// TIA Portal V19 export
FUNCTION "Flowmeter Diag" : Void   // FC10, LAD
{ S7_Optimized_Access := 'TRUE' }
// stored: SetENOAutomatically false
BEGIN

REGION Network 1
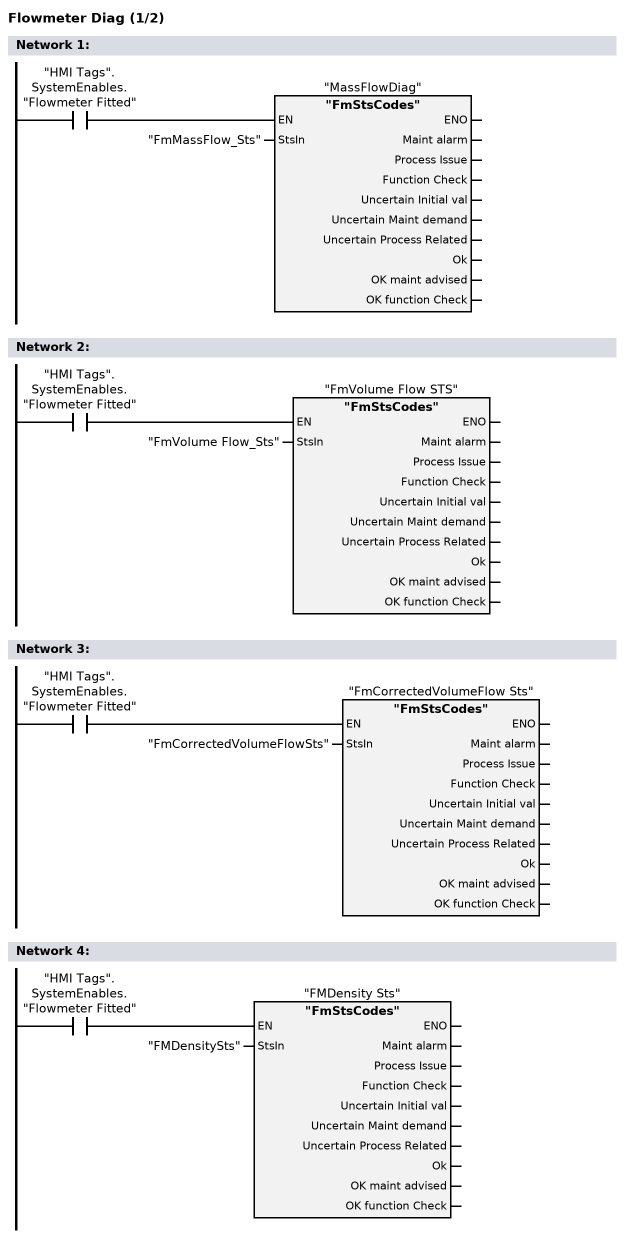
   RUNG wire#powerrail
      Contact( "HMI Tags".SystemEnables."Flowmeter Fitted" )
      "MassFlowDiag"(StsIn := "FmMassFlow_Sts", "Maint alarm" =>, "Process Issue" =>, "Function Check" =>, "Uncertain Initial val" =>, "Uncertain Maint demand" =>, "Uncertain Process Related" =>, Ok =>, "OK maint advised" =>, "OK function Check" =>)
   END_RUNG
   // the same network as SCL:
   IF "HMI Tags".SystemEnables."Flowmeter Fitted" THEN
       "MassFlowDiag"(StsIn := "FmMassFlow_Sts");   // "FmStsCodes"
   END_IF;
END_REGION

REGION Network 2
   RUNG wire#powerrail
      Contact( "HMI Tags".SystemEnables."Flowmeter Fitted" )
      "FmVolume Flow STS"(StsIn := "FmVolume Flow_Sts", "Maint alarm" =>, "Process Issue" =>, "Function Check" =>, "Uncertain Initial val" =>, "Uncertain Maint demand" =>, "Uncertain Process Related" =>, Ok =>, "OK maint advised" =>, "OK function Check" =>)
   END_RUNG
   // the same network as SCL:
   IF "HMI Tags".SystemEnables."Flowmeter Fitted" THEN
       "FmVolume Flow STS"(StsIn := "FmVolume Flow_Sts");   // "FmStsCodes"
   END_IF;
END_REGION

REGION Network 3
   RUNG wire#powerrail
      Contact( "HMI Tags".SystemEnables."Flowmeter Fitted" )
      "FmCorrectedVolumeFlow Sts"(StsIn := "FmCorrectedVolumeFlowSts", "Maint alarm" =>, "Process Issue" =>, "Function Check" =>, "Uncertain Initial val" =>, "Uncertain Maint demand" =>, "Uncertain Process Related" =>, Ok =>, "OK maint advised" =>, "OK function Check" =>)
   END_RUNG
   // the same network as SCL:
   IF "HMI Tags".SystemEnables."Flowmeter Fitted" THEN
       "FmCorrectedVolumeFlow Sts"(StsIn := "FmCorrectedVolumeFlowSts");   // "FmStsCodes"
   END_IF;
END_REGION

REGION Network 4
   RUNG wire#powerrail
      Contact( "HMI Tags".SystemEnables."Flowmeter Fitted" )
      "FMDensity Sts"(StsIn := "FMDensitySts", "Maint alarm" =>, "Process Issue" =>, "Function Check" =>, "Uncertain Initial val" =>, "Uncertain Maint demand" =>, "Uncertain Process Related" =>, Ok =>, "OK maint advised" =>, "OK function Check" =>)
   END_RUNG
   // the same network as SCL:
   IF "HMI Tags".SystemEnables."Flowmeter Fitted" THEN
       "FMDensity Sts"(StsIn := "FMDensitySts");   // "FmStsCodes"
   END_IF;
END_REGION

REGION Network 5
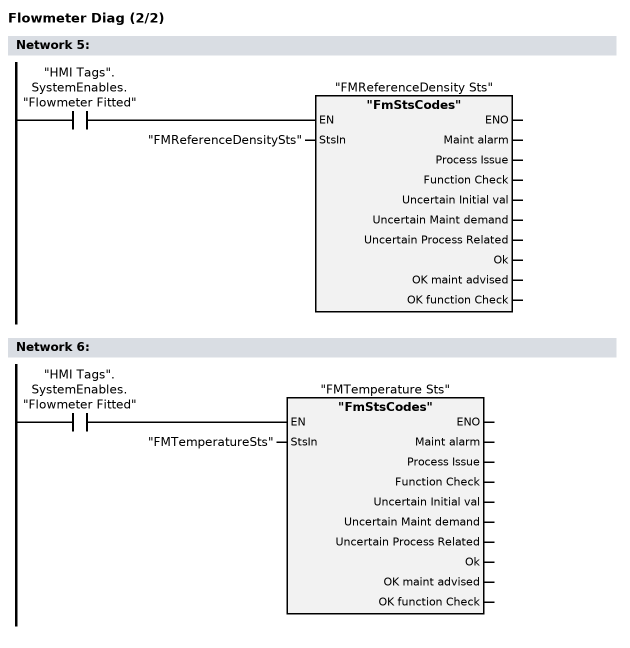
   RUNG wire#powerrail
      Contact( "HMI Tags".SystemEnables."Flowmeter Fitted" )
      "FMReferenceDensity Sts"(StsIn := "FMReferenceDensitySts", "Maint alarm" =>, "Process Issue" =>, "Function Check" =>, "Uncertain Initial val" =>, "Uncertain Maint demand" =>, "Uncertain Process Related" =>, Ok =>, "OK maint advised" =>, "OK function Check" =>)
   END_RUNG
   // the same network as SCL:
   IF "HMI Tags".SystemEnables."Flowmeter Fitted" THEN
       "FMReferenceDensity Sts"(StsIn := "FMReferenceDensitySts");   // "FmStsCodes"
   END_IF;
END_REGION

REGION Network 6
   RUNG wire#powerrail
      Contact( "HMI Tags".SystemEnables."Flowmeter Fitted" )
      "FMTemperature Sts"(StsIn := "FMTemperatureSts", "Maint alarm" =>, "Process Issue" =>, "Function Check" =>, "Uncertain Initial val" =>, "Uncertain Maint demand" =>, "Uncertain Process Related" =>, Ok =>, "OK maint advised" =>, "OK function Check" =>)
   END_RUNG
   // the same network as SCL:
   IF "HMI Tags".SystemEnables."Flowmeter Fitted" THEN
       "FMTemperature Sts"(StsIn := "FMTemperatureSts");   // "FmStsCodes"
   END_IF;
END_REGION
END_FUNCTION
